// TIA Portal V20 export
// export: Created 2026-04-11T06:02:29.980725Z, ExportSetting WithDefaults, DisplayName Totally Integrated Automation Portal, DisplayVersion V20, DisplayName TIA Portal Openness, DisplayVersion V20, DisplayName TIA Portal Version Control Interface, DisplayVersion V20, DisplayName STEP 7 Professional, DisplayVersion V20, DisplayName STEP 7 Safety, DisplayVersion V20, DisplayName WinCC Basic/Comfort/Advanced, DisplayVersion V20, DisplayName WinCC Unified, DisplayVersion V20
TYPE "udtError_AnalogValve"
// stored: IsFailsafeCompliant false
   STRUCT
      InvalidFeedback { ExternalWritable := 'False'} : Bool;   // Valve feedback is not within command tolerance
   END_STRUCT;
END_TYPE
